FUNCTION_BLOCK SUBSCRIBE_0
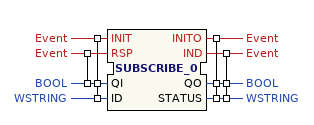
  EVENT_INPUT
    INIT WITH QI, ID;
    RSP WITH QI;
  END_EVENT
  EVENT_OUTPUT
    INITO WITH QO, STATUS;
    IND WITH QO, STATUS;
  END_EVENT
  VAR_INPUT
    QI : BOOL;
    ID : WSTRING;
  END_VAR
  VAR_OUTPUT
    QO : BOOL;
    STATUS : WSTRING;
  END_VAR
END_FUNCTION_BLOCK
